(* IEC 61131-3 sources: AXOpen/src/core/ctrl/src/AxoContext, 2 files *)

(* ---- AxoContext.st ---- *)
USING AXOpen.Messaging;
USING AXOpen.Rtc;
USING AXOpen.Logging;
USING AXOpen.Rtm;

NAMESPACE AXOpen.Core
    ///<summary>
    /// Provides base for contextualized entry of `AXOpen` application.
    /// This class is abstract and must be inherited.
    ///</summary>
    {S7.extern=ReadWrite}
    CLASS PUBLIC ABSTRACT AxoContext IMPLEMENTS IAxoContext
        VAR PRIVATE
            _openCounter : ULINT;
            _closeCounter : ULINT;
            _identityCounter : ULINT;
         END_VAR

        ///<summary>
        /// The entry point for the context. The call tree of the context start here and all the logic of given context
        /// must be placed here.
        /// This method must be overridden in derived class.
        ///</summary>
        METHOD PROTECTED ABSTRACT Main END_METHOD

        METHOD PRIVATE Open : ULINT
            _openCounter := _openCounter + ULINT#1;
        END_METHOD

        METHOD PRIVATE Close : ULINT
            _closeCounter := _closeCounter + ULINT#1;
        END_METHOD

        ///<summary>
        /// Runs the cycle of this context. This method must be called cyclically in a PLC task.
        ///</summary>
        METHOD PUBLIC Run
            THIS.Open();
            THIS.Main();
            THIS.Close();
        END_METHOD

        ///<summary>
        /// Gets the value of current context cycle counter.
        ///</summary>
        METHOD PUBLIC OpenCycleCount : ULINT
            OpenCycleCount := _openCounter;
        END_METHOD

        METHOD PUBLIC ClosedCycleCount : ULINT
            ClosedCycleCount := _closeCounter;
        END_METHOD

        METHOD PUBLIC CreateIdentity : ULINT
            _identityCounter := _identityCounter + ULINT#1;
            CreateIdentity := _identityCounter;
        END_METHOD

        METHOD PUBLIC PeekIdentity : ULINT
            PeekIdentity := _identityCounter;
        END_METHOD

        VAR PRIVATE
            NULL_RTC : _NULL_RTC;
            _rtc : IAxoRtc;
        END_VAR

        METHOD PUBLIC GetRtc : IAxoRtc
            IF(_rtc <> NULL) THEN
                GetRtc := _rtc;
            ELSE
                GetRtc := NULL_RTC;
            END_IF;
        END_METHOD

        METHOD PUBLIC InjectRtc
            VAR_INPUT
                Rtc : IAxoRtc;
            END_VAR
            _rtc := Rtc;
        END_METHOD

        VAR PRIVATE
            NULL_RTM : _NULL_RTM;
            _rtm : IAxoRtm;
        END_VAR

        METHOD PUBLIC InjectRtm
            VAR_INPUT
                inRtm : IAxoRtm;
            END_VAR
            _rtm := inRtm;
        END_METHOD

        METHOD PUBLIC GetRtm : IAxoRtm
            IF(_rtc <> NULL) THEN
                GetRtm := _rtm;
            ELSE
                GetRtm := NULL_RTM;
            END_IF;
        END_METHOD

        VAR PRIVATE
            NULL_LOGGER : _NULL_LOGGER;
            _contextLogger : IAxoLogger;
        END_VAR

        METHOD PUBLIC GetLogger : IAxoLogger
            IF(_contextLogger <> NULL) THEN
                GetLogger := _contextLogger;
            ELSE
                GetLogger := NULL_LOGGER;
            END_IF;
        END_METHOD

        METHOD PUBLIC InjectLogger
            VAR_INPUT
                _logger : IAxoLogger;
            END_VAR
            _contextLogger := _logger;
        END_METHOD
    END_CLASS
END_NAMESPACE

(* ---- AxoContextEnvironment.st ---- *)
USING AXOpen.Messaging;

NAMESPACE AXOpen.Core
    CLASS PUBLIC AxoContextEnvironment IMPLEMENTS IAxoContextEnvironment
        VAR PRIVATE
            _messenger : AxoMessengerEnv;
        END_VAR
        METHOD PUBLIC Messaging : IAxoMessengerEnv
            Messaging := _messenger;
        END_METHOD
    END_CLASS
END_NAMESPACE
